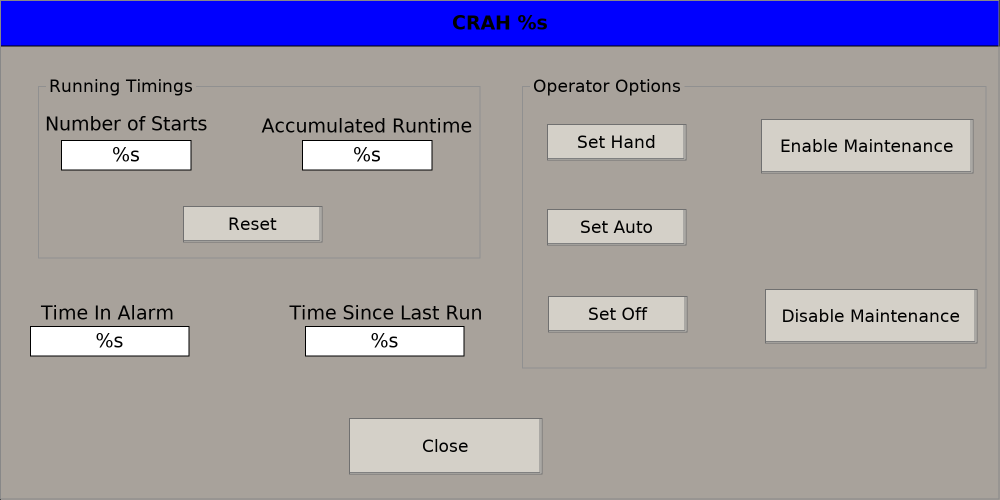
VISUALIZATION Dialog_CRAH  // 1000x500
VAR_IN_OUT
	sHeader : WSTRING;
	bCommonAlarm : BOOL;
	bIsolator1Alm :BOOL;
	bIsolator2Alm :BOOL;
	nSetControl :WORD;
	iNumStarts : WORD;
	sAccTime : STRING;
	sAlarmTime : STRING;
	sLastRunTime : STRING;
	bSetMaintenance : BOOL;
	bResetTimings : BOOL;
END_VAR
    GroupBox (38,78 442x180), "Running Timings"
        Button (145,128 139x36), "Reset"
            OnMouseClick: execute { bResetTimings:=1; }
    Rectangle (0,0 1000x46), "CRAH %s", text variable: sHeader
    Label (29,298 157x30), "Time In Alarm"
    Rectangle (30,326 159x30), "%s", text variable: sAlarmTime
    Label (39,109 175x30), "Number of Starts"
    Rectangle (61,140 130x30), "%s", text variable: iNumStarts
    Label (257,111 220x30), "Accumulated Runtime"
    Rectangle (302,140 130x30), "%s", text variable: sAccTime
    Label (285,298 202x30), "Time Since Last Run"
    Rectangle (305,326 159x30), "%s", text variable: sLastRunTime
    GroupBox (522,78 464x290), "Operator Options"
        Button (25,46 139x36), "Set Hand"
            OnMouseClick: execute { nSetControl:= 0; }
            OnMouseClick: CloseDialog Dialog=Dialog_CRAH, Result=OK, NumpadKeypadSet=True
        Button (25,131 139x36), "Set Auto"
            OnMouseClick: execute { nSetControl:= 2; }
            OnMouseClick: CloseDialog Dialog=Dialog_CRAH, Result=OK, NumpadKeypadSet=True
        Button (26,218 139x36), "Set Off"
            OnMouseClick: execute { nSetControl:= 1; }
            OnMouseClick: CloseDialog Dialog=Dialog_CRAH, Result=OK, NumpadKeypadSet=True
        Button (239,41 212x54), "Enable Maintenance"
            OnMouseClick: execute { bSetMaintenance:= 1; }
            OnMouseClick: CloseDialog Dialog=Dialog_CRAH, Result=OK, NumpadKeypadSet=True
        Button (243,211 212x54), "Disable Maintenance"
            OnMouseClick: execute { bSetMaintenance:= 0; }
            OnMouseClick: CloseDialog Dialog=Dialog_CRAH, Result=OK, NumpadKeypadSet=True
    Button (349,418 193x56), "Close"
        OnMouseClick: CloseDialog Dialog=Dialog_CRAH, Result=OK, NumpadKeypadSet=True
    Line (1000,0) (1000,500)
    Line (0,0) (0,500)
    Line (0,500) (1000,500)
END_VISUALIZATION

(* stored: Version 1.1.0.1, ProductVersion 3.1.4024.12
   Visu Dialog_CRAH: Id {e26929d1-4c9c-4902-bbb0-f35292e44841} *)
